Omron CX-Programmer project NewProject (CX-Programmer 9.73)

# PLC NewPLC1: C200HS CPU01

## Program NewProgram1 (no task)
; 欧姆龙电镀控制系统。 系统通过启动按钮启动工作流程，控制加热器、搅拌器和电镀电源，并包含故障检测和保护功能。 / 项目使用的物理设备包括PLC控制器、启动按钮、停止按钮、手动/自动开关、加热器、搅拌器、电镀电源、温度传感器、液位传感器、电流传感器和报警灯。 / 系统配备启动按钮、停止按钮和手动/自动切换开关。 / 在自动模式下，启动按钮触发系统运行。只有在停止按钮未按下时，系统才能启动，同时模式信号表示系统处于自动运行状态。 / 系统启动后，加热器开始工作。 / 搅拌器启动后，利用搅拌延时定时器 (TIM492) 控制搅拌时间。 / 电镀电源启动后，由电镀延时定时器 (TIM499) 控制电镀时长。 / 系统运行期间，监控关键参数。电流传感器将检测值与安全上限进行比较。液位传感器将检测值与安全下限进行比较。 / 当温度传感器检测到温度超出安全范围时，报警灯亮起。当电流传感器检测到电流超过安全上限时，报警灯亮起。当液位传感器检测到液位低于安全下限时，报警灯亮起。报警信号用于记录系统异常状态。 / 在手动模式下，操作员可控制设备。 / 实际应用中，该系统部署在电镀车间，使用的物理设备包括PLC控制器C200HS CPU01、启动按钮、停止按钮、手动/自动切换开关、加热器、搅拌器、电镀电源，以及温度传感器、液位传感器、电流传感器和报警灯。 / 为确保系统稳定运行，维护人员需定期检查温度传感器、液位传感器和电流传感器的工作状态，确认手动/自动切换开关切换正常，验证搅拌延时定时器 (TIM492) 和电镀延时定时器 (TIM499) 的时间设置是否准确，并通过观察报警灯的状态及时响应异常情况。 / 程序以END指令结束扫描周期，确保每次运行逻辑清晰可控。

### Section Section1

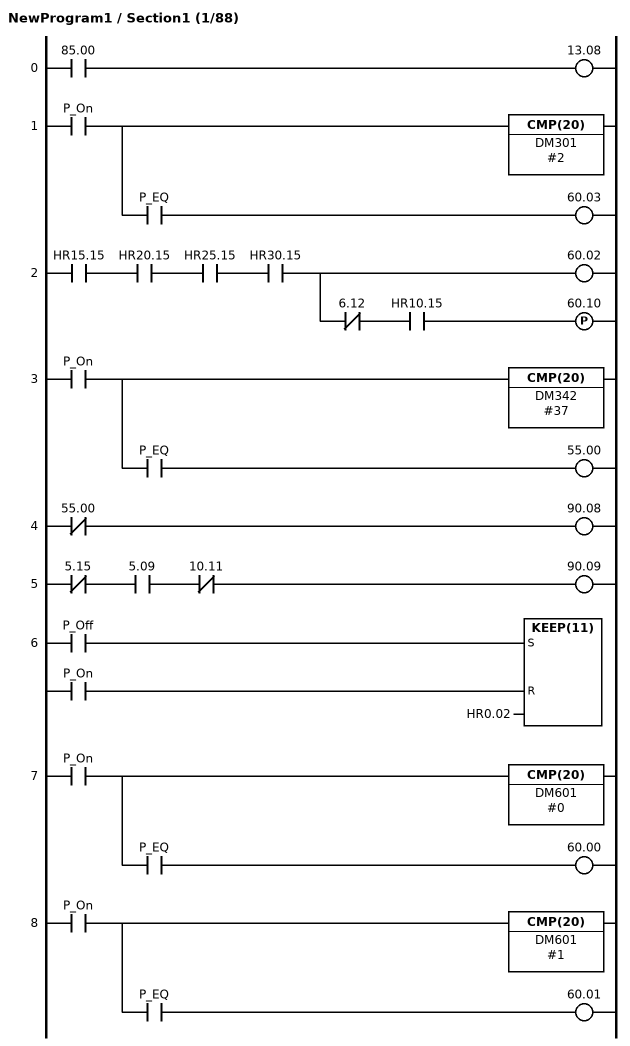
; rung 0
LD 85.00
OUT 13.08
; rung 1
LD P_On
CMP(20) DM301 #2
AND P_EQ
OUT 60.03
; rung 2
LD HR15.15
AND HR20.15
AND HR25.15
AND HR30.15
OUT 60.02
ANDNOT 6.12
AND HR10.15
DIFU(13) 60.10
; rung 3
LD P_On
CMP(20) DM342 #37
AND P_EQ
OUT 55.00
; rung 4
LDNOT 55.00
OUT 90.08
; rung 5
LDNOT 5.15
AND 5.09
ANDNOT 10.11
OUT 90.09
; rung 6
LD P_Off
LD P_On
KEEP(11) HR0.02
; rung 7
LD P_On
CMP(20) DM601 #0
AND P_EQ
OUT 60.00
; rung 8
LD P_On
CMP(20) DM601 #1
AND P_EQ
OUT 60.01

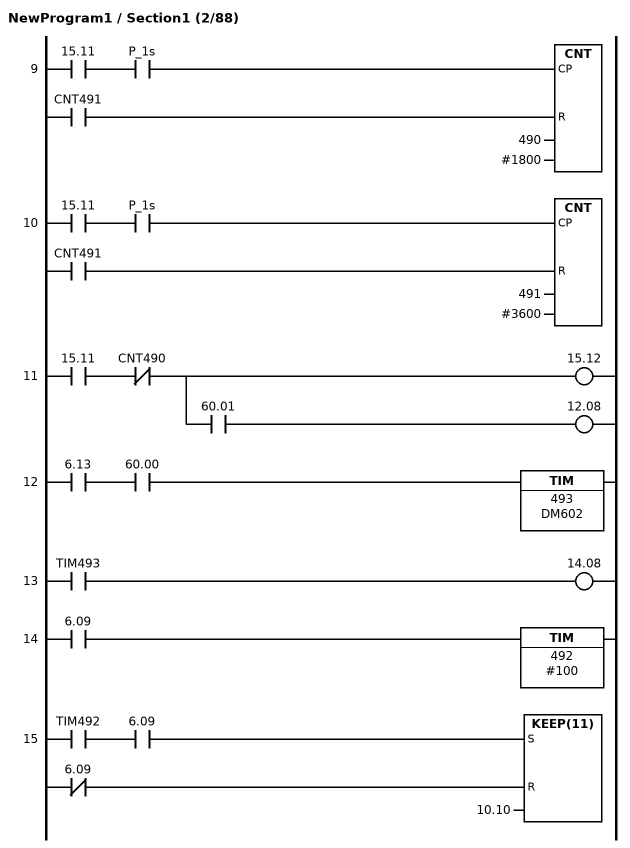
; rung 9
LD 15.11
AND P_1s
LD CNT491
CNT 490 #1800
; rung 10
LD 15.11
AND P_1s
LD CNT491
CNT 491 #3600
; rung 11
LD 15.11
ANDNOT CNT490
OUT 15.12
AND 60.01
OUT 12.08
; rung 12
LD 6.13
AND 60.00
TIM 493 DM602
; rung 13
LD TIM493
OUT 14.08
; rung 14
LD 6.09
TIM 492 #100
; rung 15
LD TIM492
AND 6.09
LDNOT 6.09
KEEP(11) 10.10

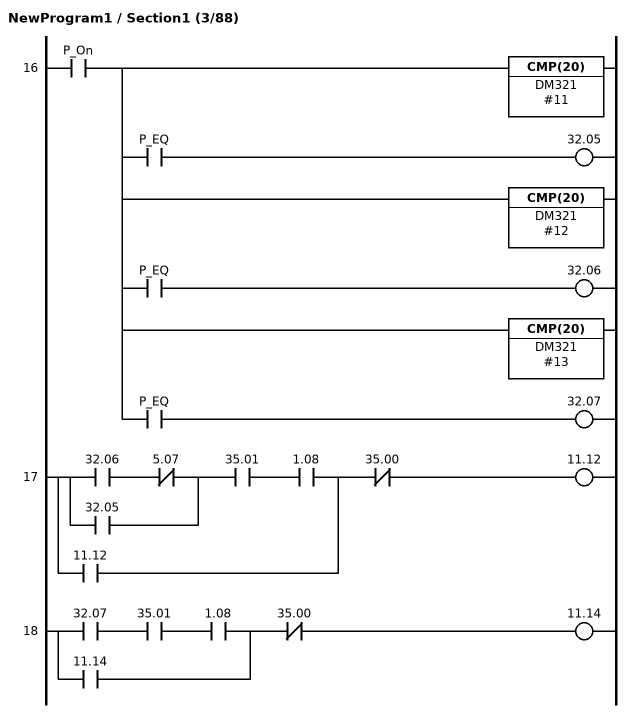
; rung 16
LD P_On
OUT TR0
CMP(20) DM321 #11
AND P_EQ
OUT 32.05
LD TR0
CMP(20) DM321 #12
AND P_EQ
OUT 32.06
LD TR0
CMP(20) DM321 #13
AND P_EQ
OUT 32.07
; rung 17
LD 32.06
ANDNOT 5.07
OR 32.05
AND 35.01
AND 1.08
OR 11.12
ANDNOT 35.00
OUT 11.12
; rung 18
LD 32.07
AND 35.01
AND 1.08
OR 11.14
ANDNOT 35.00
OUT 11.14

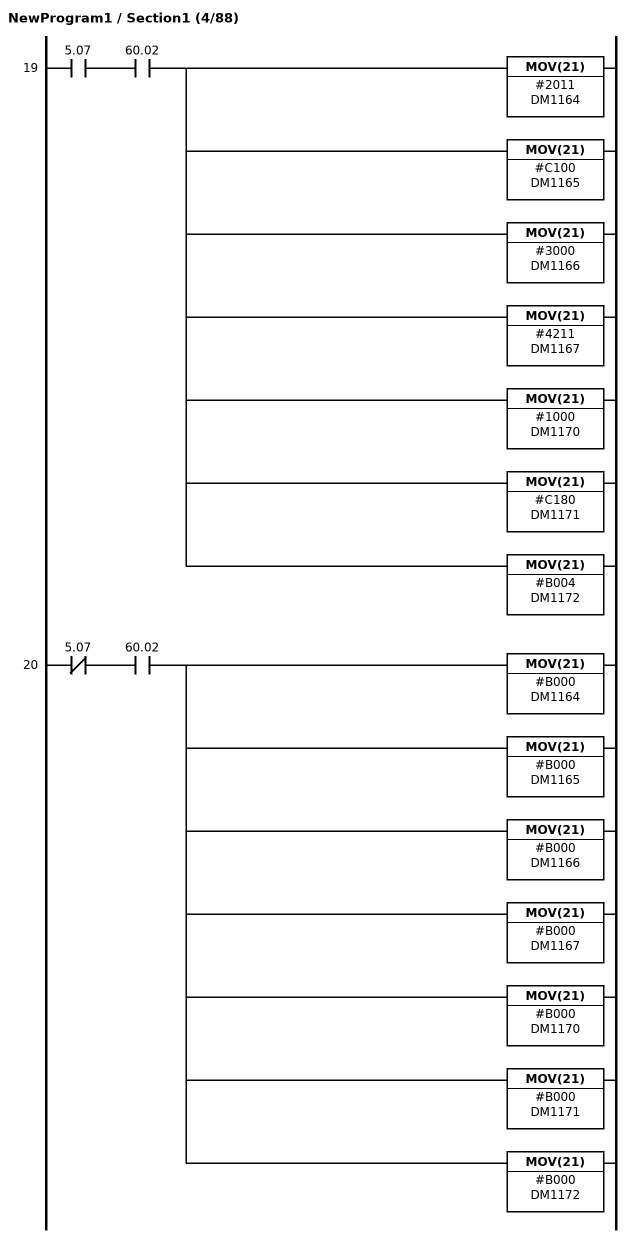
; rung 19
LD 5.07
AND 60.02
MOV(21) #2011 DM1164
MOV(21) #C100 DM1165
MOV(21) #3000 DM1166
MOV(21) #4211 DM1167
MOV(21) #1000 DM1170
MOV(21) #C180 DM1171
MOV(21) #B004 DM1172
; rung 20
LDNOT 5.07
AND 60.02
MOV(21) #B000 DM1164
MOV(21) #B000 DM1165
MOV(21) #B000 DM1166
MOV(21) #B000 DM1167
MOV(21) #B000 DM1170
MOV(21) #B000 DM1171
MOV(21) #B000 DM1172

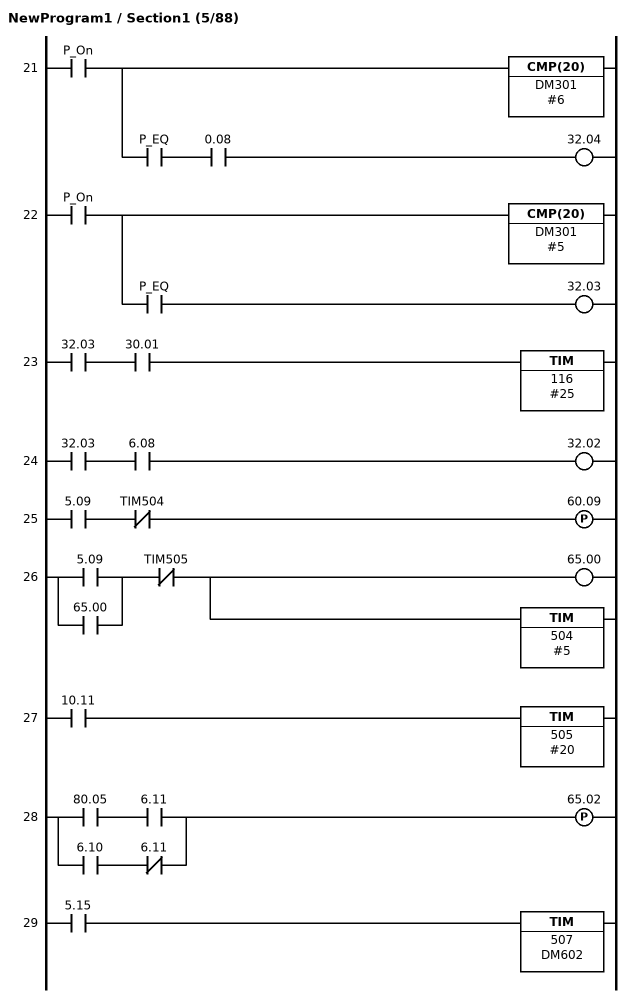
; rung 21
LD P_On
CMP(20) DM301 #6
AND P_EQ
AND 0.08
OUT 32.04
; rung 22
LD P_On
CMP(20) DM301 #5
AND P_EQ
OUT 32.03
; rung 23
LD 32.03
AND 30.01
TIM 116 #25
; rung 24
LD 32.03
AND 6.08
OUT 32.02
; rung 25
LD 5.09
ANDNOT TIM504
DIFU(13) 60.09
; rung 26
LD 5.09
OR 65.00
ANDNOT TIM505
OUT 65.00
TIM 504 #5
; rung 27
LD 10.11
TIM 505 #20
; rung 28
LD 80.05
AND 6.11
LD 6.10
ANDNOT 6.11
ORLD
DIFU(13) 65.02
; rung 29
LD 5.15
TIM 507 DM602

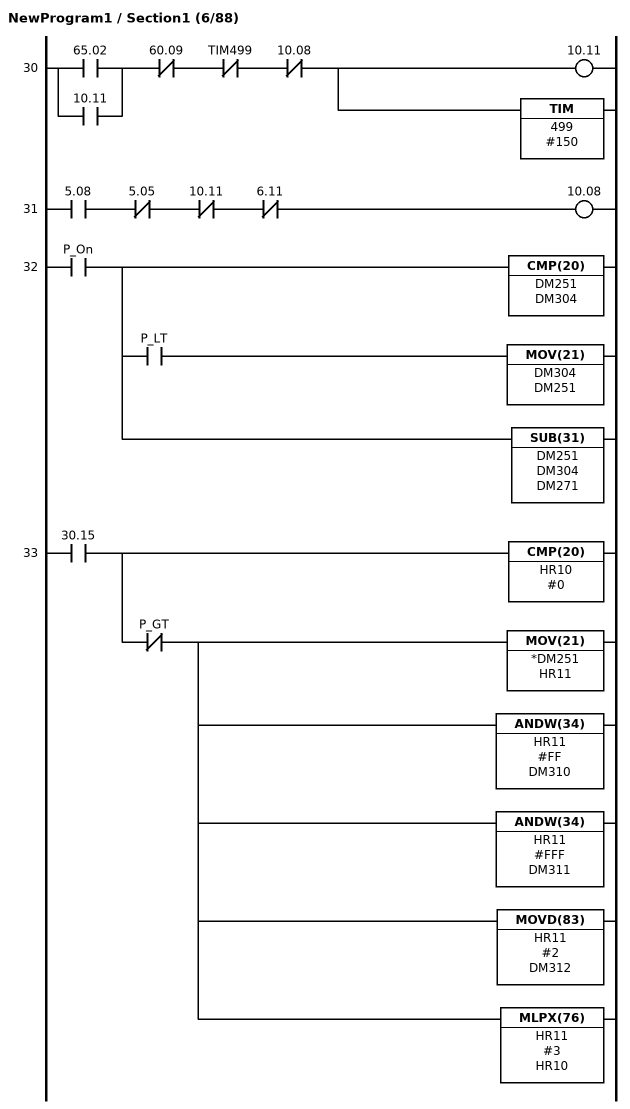
; rung 30
LD 65.02
OR 10.11
ANDNOT 60.09
ANDNOT TIM499
ANDNOT 10.08
OUT 10.11
TIM 499 #150
; rung 31
LD 5.08
ANDNOT 5.05
ANDNOT 10.11
ANDNOT 6.11
OUT 10.08
; rung 32
LD P_On
OUT TR0
CMP(20) DM251 DM304
AND P_LT
MOV(21) DM304 DM251
LD TR0
SUB(31) DM251 DM304 DM271
; rung 33
LD 30.15
CMP(20) HR10 #0
ANDNOT P_GT
MOV(21) *DM251 HR11
ANDW(34) HR11 #FF DM310
ANDW(34) HR11 #FFF DM311
MOVD(83) HR11 #2 DM312
MLPX(76) HR11 #3 HR10

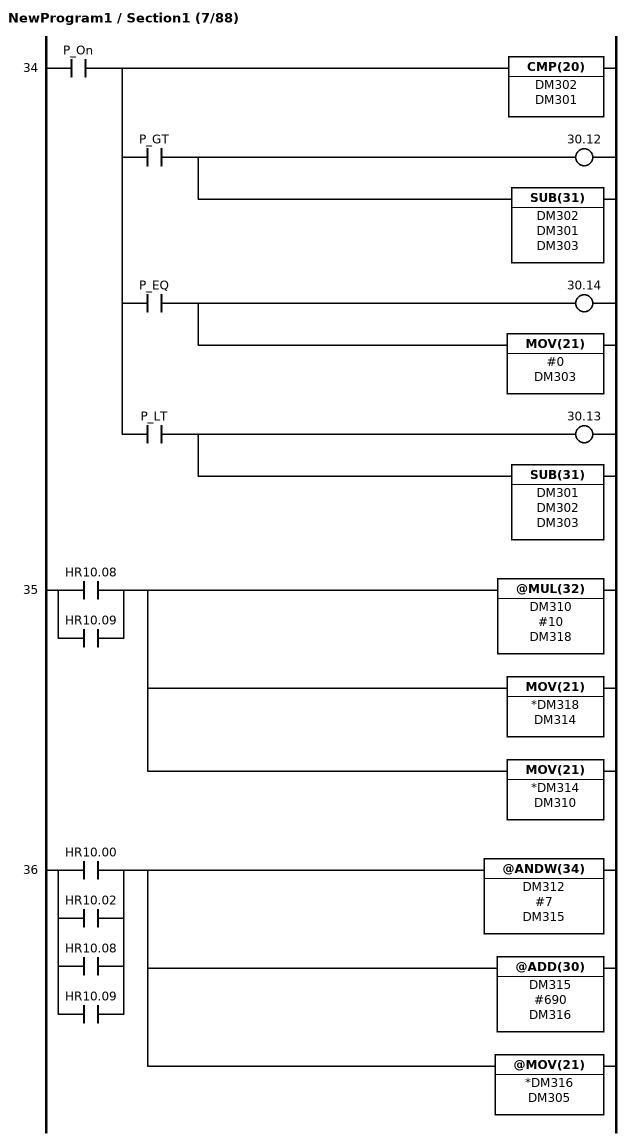
; rung 34
LD P_On
OUT TR0
CMP(20) DM302 DM301
AND P_GT
OUT 30.12
SUB(31) DM302 DM301 DM303
LD TR0
AND P_EQ
OUT 30.14
MOV(21) #0 DM303
LD TR0
AND P_LT
OUT 30.13
SUB(31) DM301 DM302 DM303
; rung 35
LD HR10.08
OR HR10.09
@MUL(32) DM310 #10 DM318
MOV(21) *DM318 DM314
MOV(21) *DM314 DM310
; rung 36
LD HR10.00
OR HR10.02
OR HR10.08
OR HR10.09
@ANDW(34) DM312 #7 DM315
@ADD(30) DM315 #690 DM316
@MOV(21) *DM316 DM305

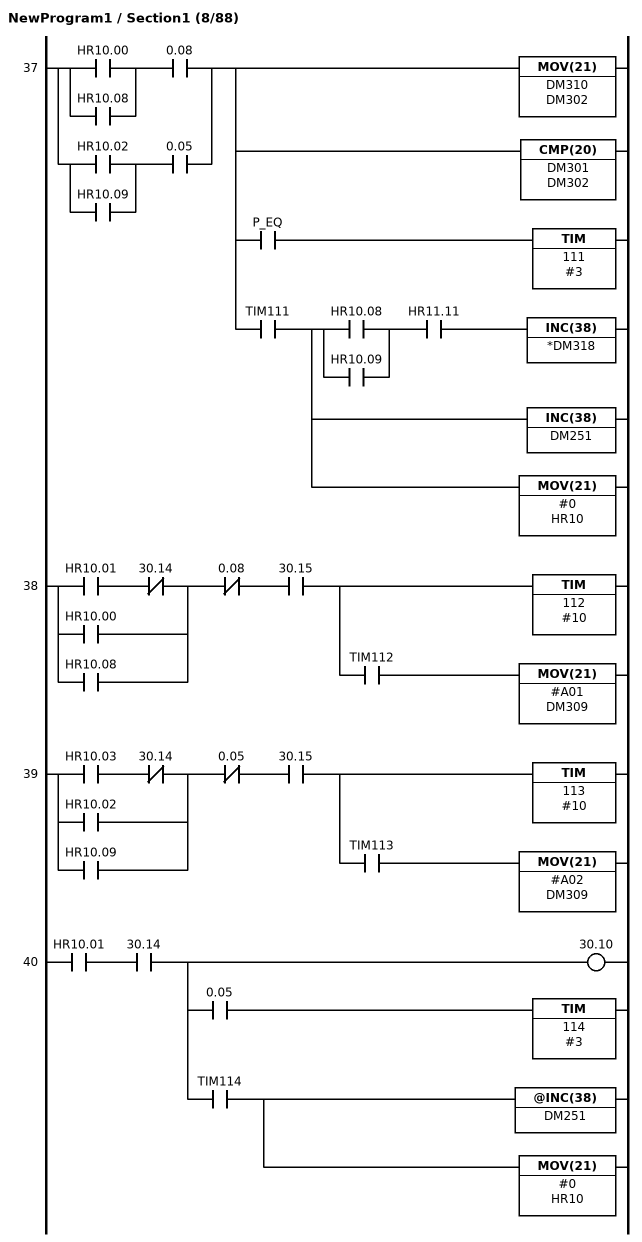
; rung 37
LD HR10.00
OR HR10.08
AND 0.08
LD HR10.02
OR HR10.09
AND 0.05
ORLD
OUT TR0
MOV(21) DM310 DM302
CMP(20) DM301 DM302
AND P_EQ
TIM 111 #3
LD TR0
AND TIM111
OUT TR0
LD HR10.08
OR HR10.09
ANDLD
AND HR11.11
INC(38) *DM318
LD TR0
INC(38) DM251
MOV(21) #0 HR10
; rung 38
LD HR10.01
ANDNOT 30.14
OR HR10.00
OR HR10.08
ANDNOT 0.08
AND 30.15
TIM 112 #10
AND TIM112
MOV(21) #A01 DM309
; rung 39
LD HR10.03
ANDNOT 30.14
OR HR10.02
OR HR10.09
ANDNOT 0.05
AND 30.15
TIM 113 #10
AND TIM113
MOV(21) #A02 DM309
; rung 40
LD HR10.01
AND 30.14
OUT TR0
OUT 30.10
AND 0.05
TIM 114 #3
LD TR0
AND TIM114
@INC(38) DM251
MOV(21) #0 HR10

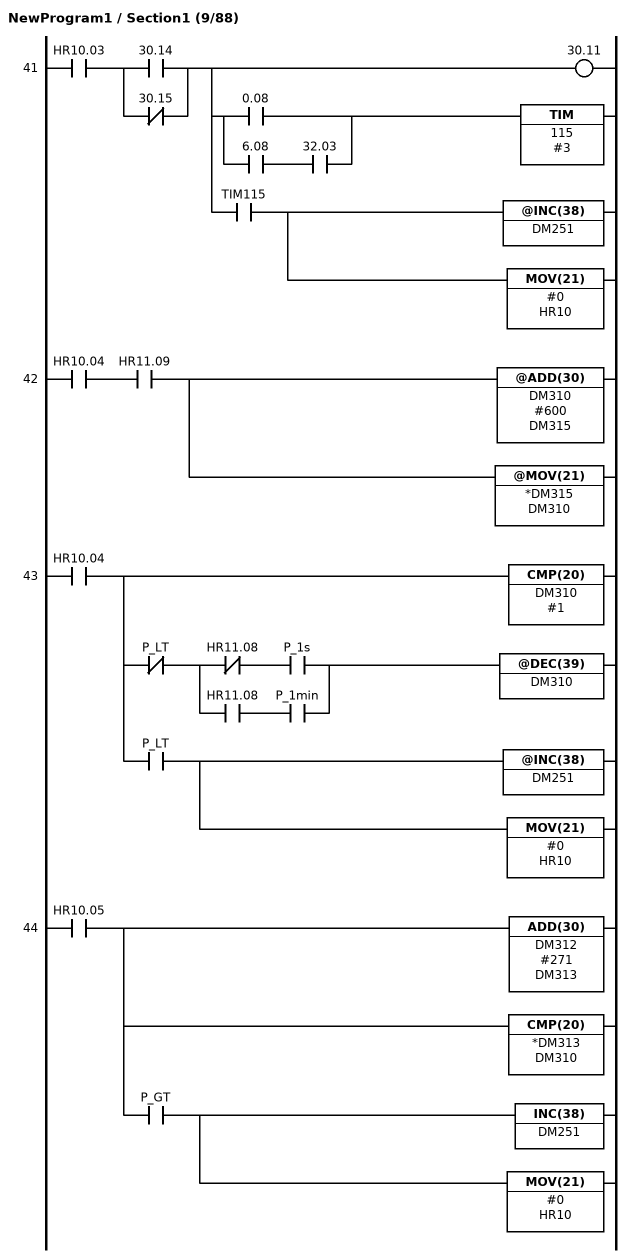
; rung 41
LD HR10.03
LD 30.14
ORNOT 30.15
ANDLD
OUT TR0
OUT 30.11
LD 0.08
LD 6.08
AND 32.03
ORLD
ANDLD
TIM 115 #3
LD TR0
AND TIM115
@INC(38) DM251
MOV(21) #0 HR10
; rung 42
LD HR10.04
AND HR11.09
@ADD(30) DM310 #600 DM315
@MOV(21) *DM315 DM310
; rung 43
LD HR10.04
OUT TR0
CMP(20) DM310 #1
ANDNOT P_LT
LDNOT HR11.08
AND P_1s
LD HR11.08
AND P_1min
ORLD
ANDLD
@DEC(39) DM310
LD TR0
AND P_LT
@INC(38) DM251
MOV(21) #0 HR10
; rung 44
LD HR10.05
ADD(30) DM312 #271 DM313
CMP(20) *DM313 DM310
AND P_GT
INC(38) DM251
MOV(21) #0 HR10

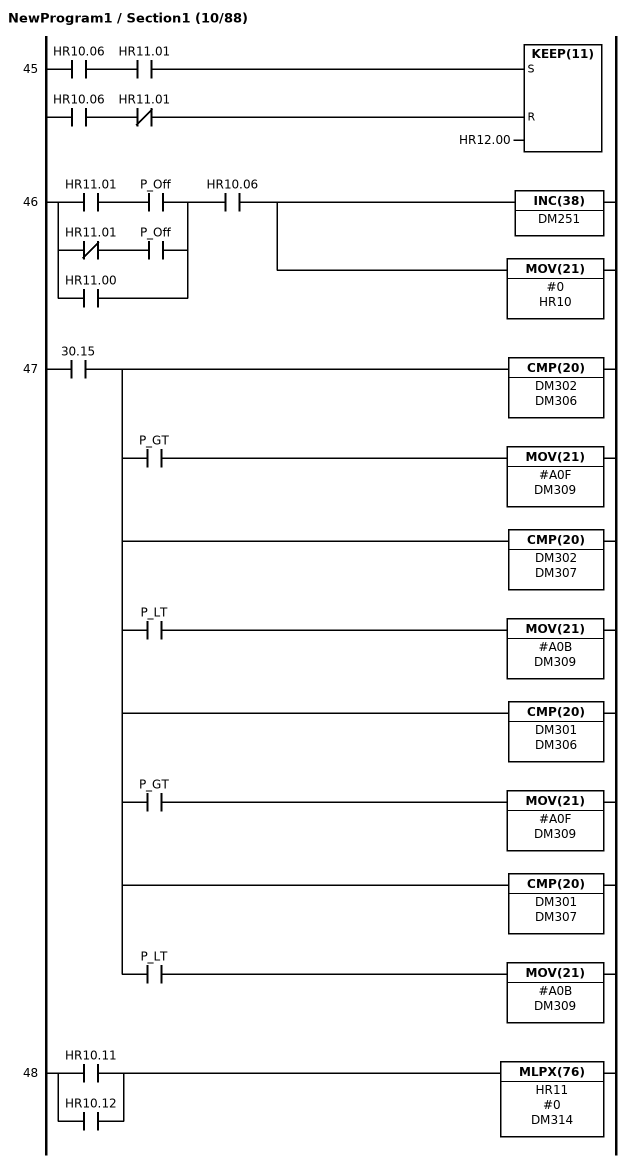
; rung 45
LD HR10.06
AND HR11.01
LD HR10.06
ANDNOT HR11.01
KEEP(11) HR12.00
; rung 46
LD HR11.01
AND P_Off
LDNOT HR11.01
AND P_Off
ORLD
OR HR11.00
AND HR10.06
INC(38) DM251
MOV(21) #0 HR10
; rung 47
LD 30.15
OUT TR0
CMP(20) DM302 DM306
AND P_GT
MOV(21) #A0F DM309
LD TR0
CMP(20) DM302 DM307
AND P_LT
MOV(21) #A0B DM309
LD TR0
CMP(20) DM301 DM306
AND P_GT
MOV(21) #A0F DM309
LD TR0
CMP(20) DM301 DM307
AND P_LT
MOV(21) #A0B DM309
; rung 48
LD HR10.11
OR HR10.12
MLPX(76) HR11 #0 DM314

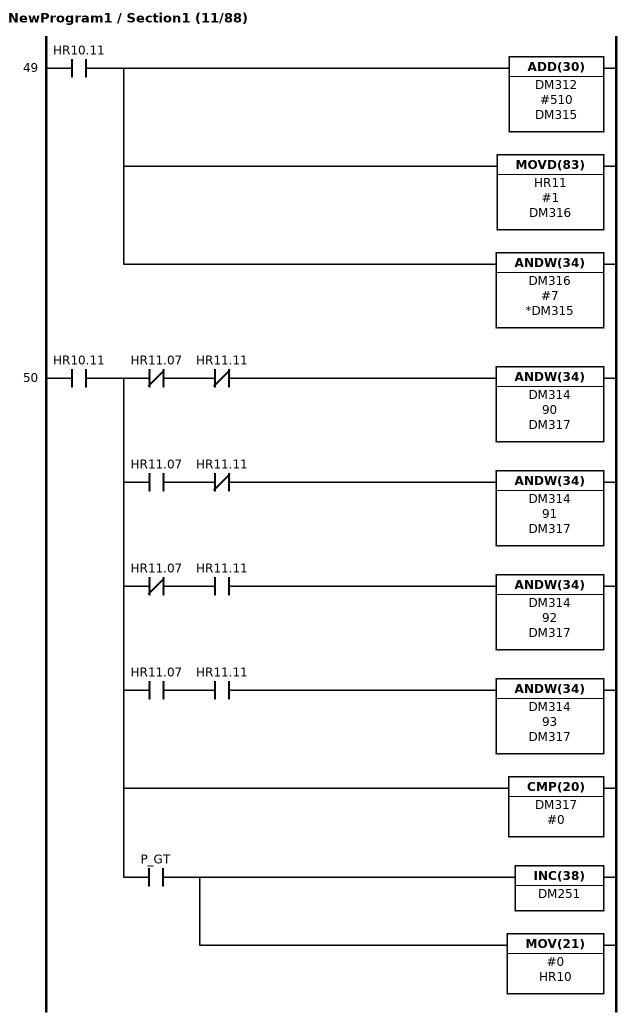
; rung 49
LD HR10.11
ADD(30) DM312 #510 DM315
MOVD(83) HR11 #1 DM316
ANDW(34) DM316 #7 *DM315
; rung 50
LD HR10.11
OUT TR0
ANDNOT HR11.07
ANDNOT HR11.11
ANDW(34) DM314 90 DM317
LD TR0
AND HR11.07
ANDNOT HR11.11
ANDW(34) DM314 91 DM317
LD TR0
ANDNOT HR11.07
AND HR11.11
ANDW(34) DM314 92 DM317
LD TR0
AND HR11.07
AND HR11.11
ANDW(34) DM314 93 DM317
LD TR0
CMP(20) DM317 #0
AND P_GT
INC(38) DM251
MOV(21) #0 HR10

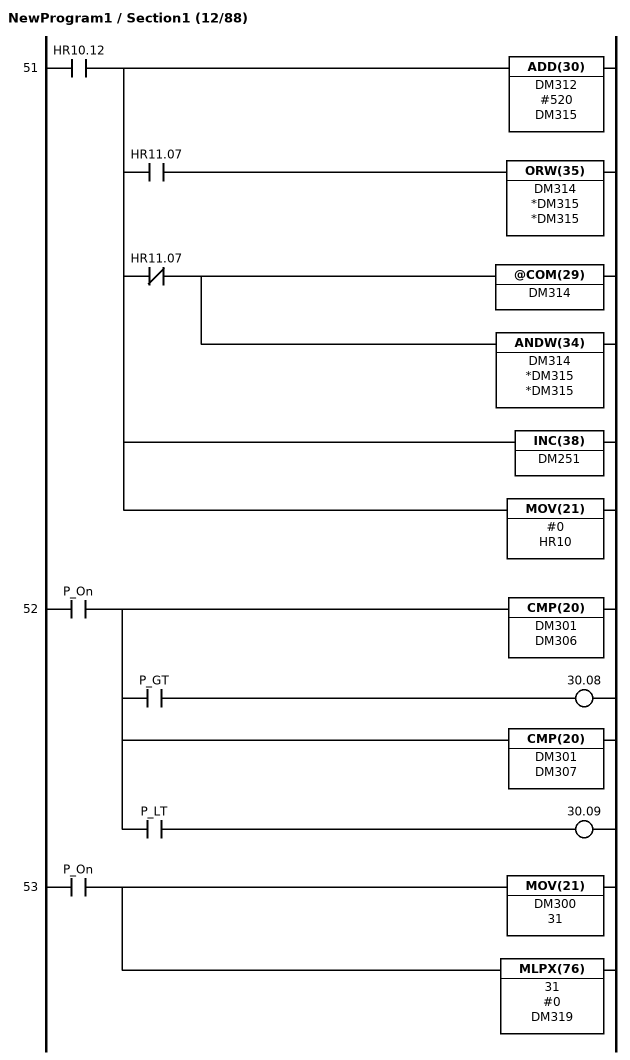
; rung 51
LD HR10.12
OUT TR0
ADD(30) DM312 #520 DM315
AND HR11.07
ORW(35) DM314 *DM315 *DM315
LD TR0
ANDNOT HR11.07
@COM(29) DM314
ANDW(34) DM314 *DM315 *DM315
LD TR0
INC(38) DM251
MOV(21) #0 HR10
; rung 52
LD P_On
OUT TR0
CMP(20) DM301 DM306
AND P_GT
OUT 30.08
LD TR0
CMP(20) DM301 DM307
AND P_LT
OUT 30.09
; rung 53
LD P_On
MOV(21) DM300 31
MLPX(76) 31 #0 DM319

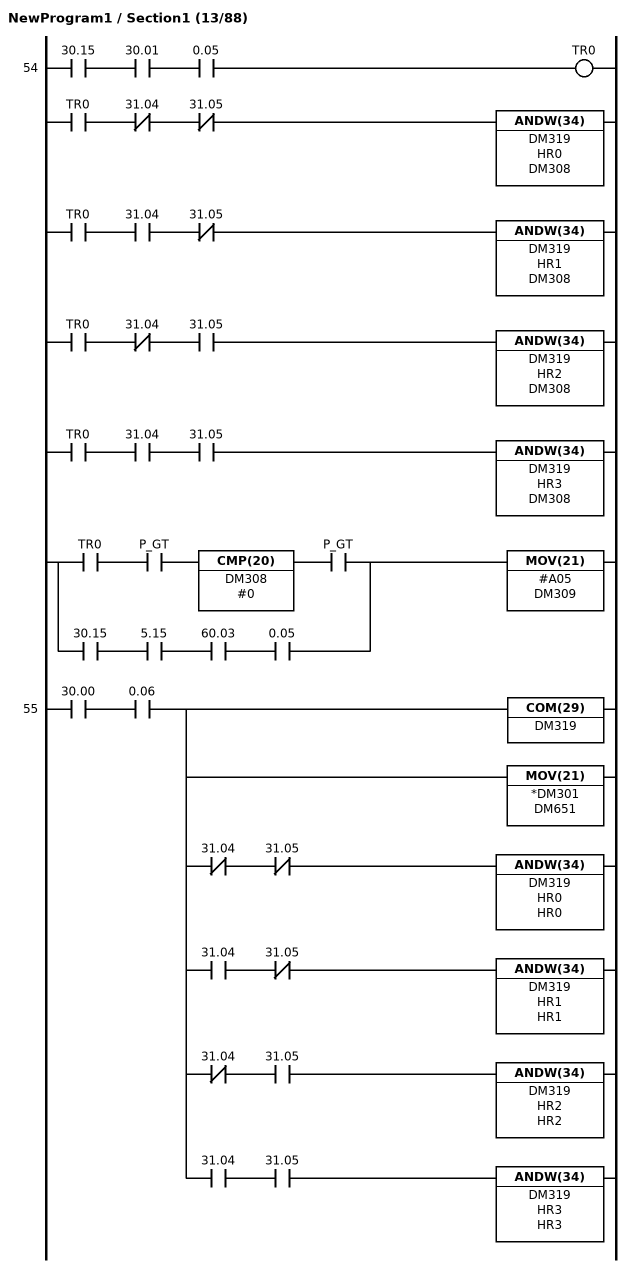
; rung 54
LD 30.15
AND 30.01
AND 0.05
OUT TR0
ANDNOT 31.04
ANDNOT 31.05
ANDW(34) DM319 HR0 DM308
LD TR0
AND 31.04
ANDNOT 31.05
ANDW(34) DM319 HR1 DM308
LD TR0
ANDNOT 31.04
AND 31.05
ANDW(34) DM319 HR2 DM308
LD TR0
AND 31.04
AND 31.05
ANDW(34) DM319 HR3 DM308
LD TR0
AND P_GT
CMP(20) DM308 #0
AND P_GT
LD 30.15
AND 5.15
AND 60.03
AND 0.05
ORLD
MOV(21) #A05 DM309
; rung 55
LD 30.00
AND 0.06
OUT TR0
COM(29) DM319
MOV(21) *DM301 DM651
ANDNOT 31.04
ANDNOT 31.05
ANDW(34) DM319 HR0 HR0
LD TR0
AND 31.04
ANDNOT 31.05
ANDW(34) DM319 HR1 HR1
LD TR0
ANDNOT 31.04
AND 31.05
ANDW(34) DM319 HR2 HR2
LD TR0
AND 31.04
AND 31.05
ANDW(34) DM319 HR3 HR3

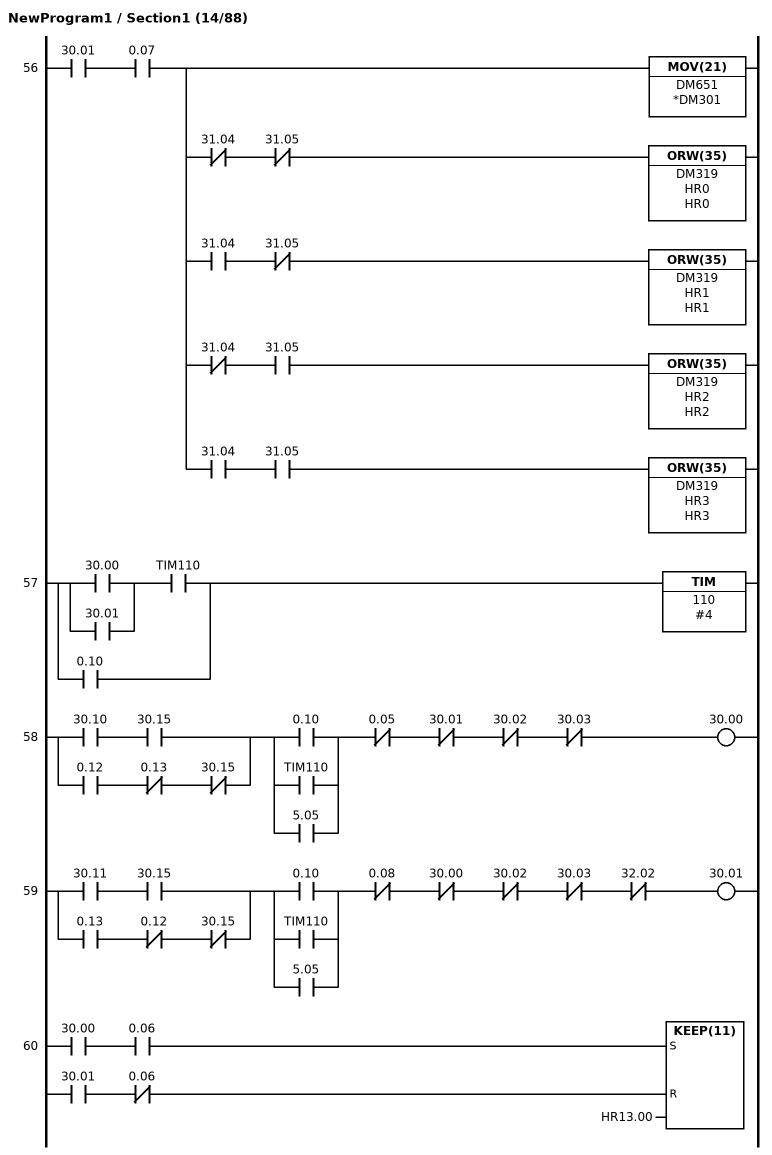
; rung 56
LD 30.01
AND 0.07
OUT TR0
MOV(21) DM651 *DM301
ANDNOT 31.04
ANDNOT 31.05
ORW(35) DM319 HR0 HR0
LD TR0
AND 31.04
ANDNOT 31.05
ORW(35) DM319 HR1 HR1
LD TR0
ANDNOT 31.04
AND 31.05
ORW(35) DM319 HR2 HR2
LD TR0
AND 31.04
AND 31.05
ORW(35) DM319 HR3 HR3
; rung 57
LD 30.00
OR 30.01
AND TIM110
OR 0.10
TIM 110 #4
; rung 58
LD 30.10
AND 30.15
LD 0.12
ANDNOT 0.13
ANDNOT 30.15
ORLD
LD 0.10
OR TIM110
OR 5.05
ANDLD
ANDNOT 0.05
ANDNOT 30.01
ANDNOT 30.02
ANDNOT 30.03
OUT 30.00
; rung 59
LD 30.11
AND 30.15
LD 0.13
ANDNOT 0.12
ANDNOT 30.15
ORLD
LD 0.10
OR TIM110
OR 5.05
ANDLD
ANDNOT 0.08
ANDNOT 30.00
ANDNOT 30.02
ANDNOT 30.03
ANDNOT 32.02
OUT 30.01
; rung 60
LD 30.00
AND 0.06
LD 30.01
ANDNOT 0.06
KEEP(11) HR13.00

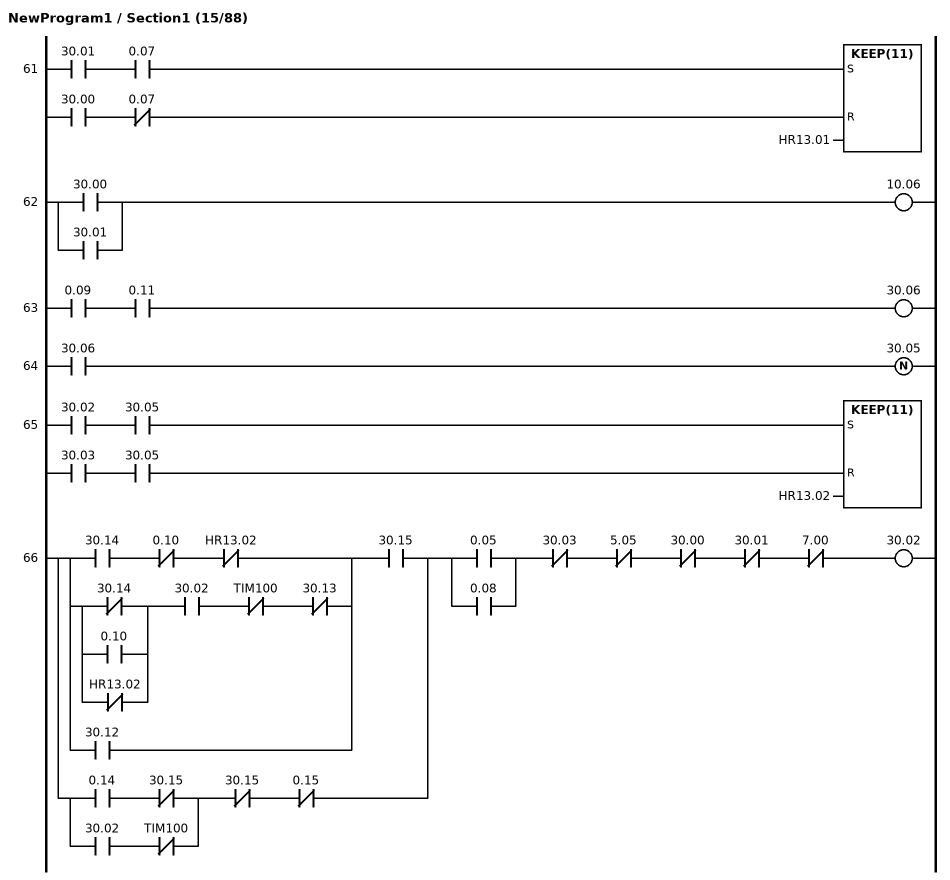
; rung 61
LD 30.01
AND 0.07
LD 30.00
ANDNOT 0.07
KEEP(11) HR13.01
; rung 62
LD 30.00
OR 30.01
OUT 10.06
; rung 63
LD 0.09
AND 0.11
OUT 30.06
; rung 64
LD 30.06
DIFD(14) 30.05
; rung 65
LD 30.02
AND 30.05
LD 30.03
AND 30.05
KEEP(11) HR13.02
; rung 66
LD 30.14
ANDNOT 0.10
ANDNOT HR13.02
LDNOT 30.14
OR 0.10
ORNOT HR13.02
AND 30.02
ANDNOT TIM100
ANDNOT 30.13
ORLD
OR 30.12
AND 30.15
LD 0.14
ANDNOT 30.15
LD 30.02
ANDNOT TIM100
ORLD
ANDNOT 30.15
ANDNOT 0.15
ORLD
LD 0.05
OR 0.08
ANDLD
ANDNOT 30.03
ANDNOT 5.05
ANDNOT 30.00
ANDNOT 30.01
ANDNOT 7.00
OUT 30.02

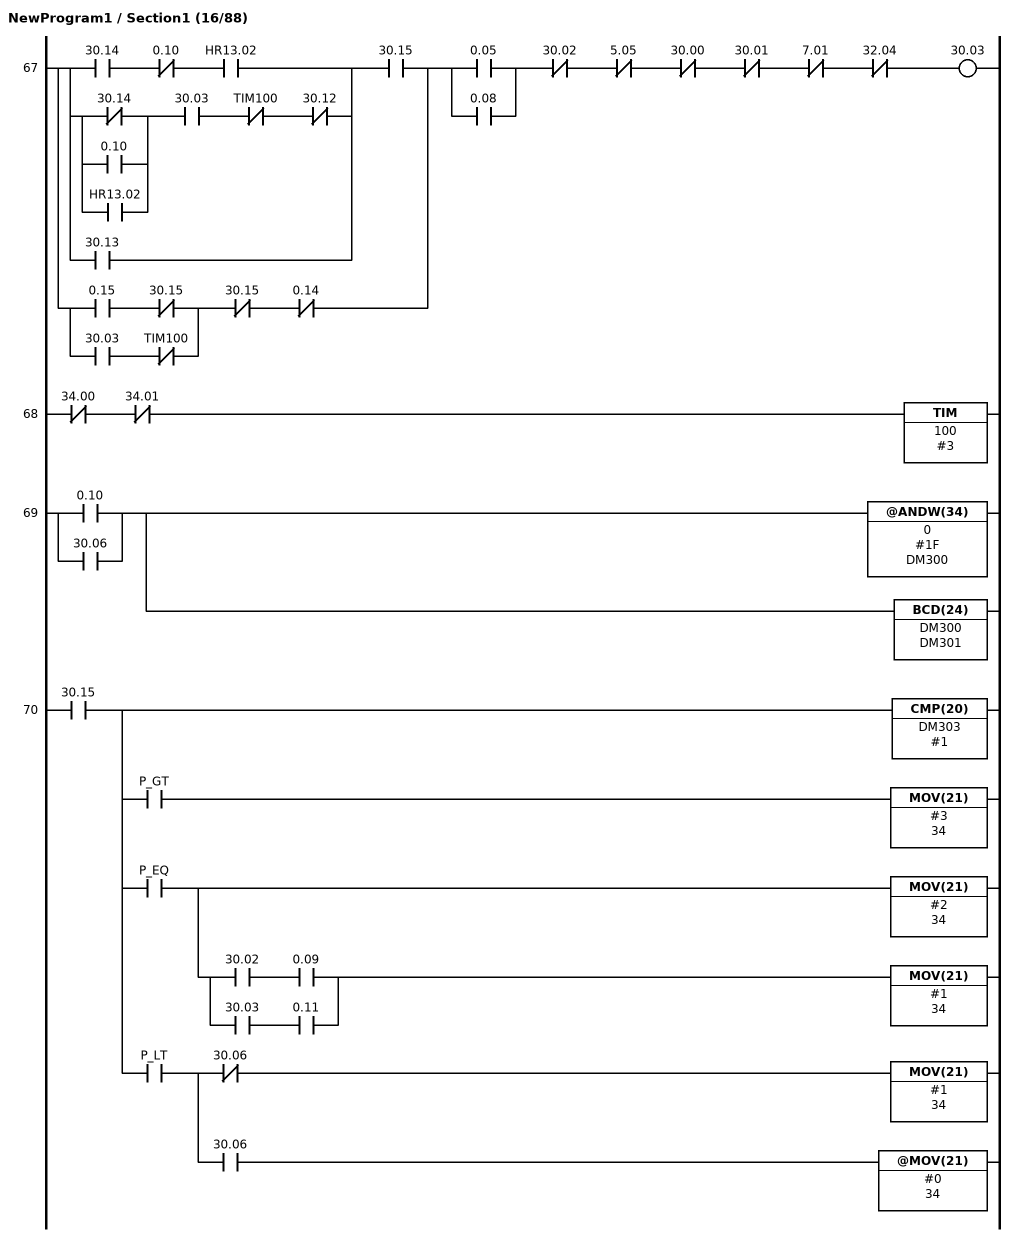
; rung 67
LD 30.14
ANDNOT 0.10
AND HR13.02
LDNOT 30.14
OR 0.10
OR HR13.02
AND 30.03
ANDNOT TIM100
ANDNOT 30.12
ORLD
OR 30.13
AND 30.15
LD 0.15
ANDNOT 30.15
LD 30.03
ANDNOT TIM100
ORLD
ANDNOT 30.15
ANDNOT 0.14
ORLD
LD 0.05
OR 0.08
ANDLD
ANDNOT 30.02
ANDNOT 5.05
ANDNOT 30.00
ANDNOT 30.01
ANDNOT 7.01
ANDNOT 32.04
OUT 30.03
; rung 68
LDNOT 34.00
ANDNOT 34.01
TIM 100 #3
; rung 69
LD 0.10
OR 30.06
@ANDW(34) 0 #1F DM300
BCD(24) DM300 DM301
; rung 70
LD 30.15
OUT TR0
CMP(20) DM303 #1
AND P_GT
MOV(21) #3 34
LD TR0
AND P_EQ
MOV(21) #2 34
LD 30.02
AND 0.09
LD 30.03
AND 0.11
ORLD
ANDLD
MOV(21) #1 34
LD TR0
AND P_LT
OUT TR0
ANDNOT 30.06
MOV(21) #1 34
LD TR0
AND 30.06
@MOV(21) #0 34

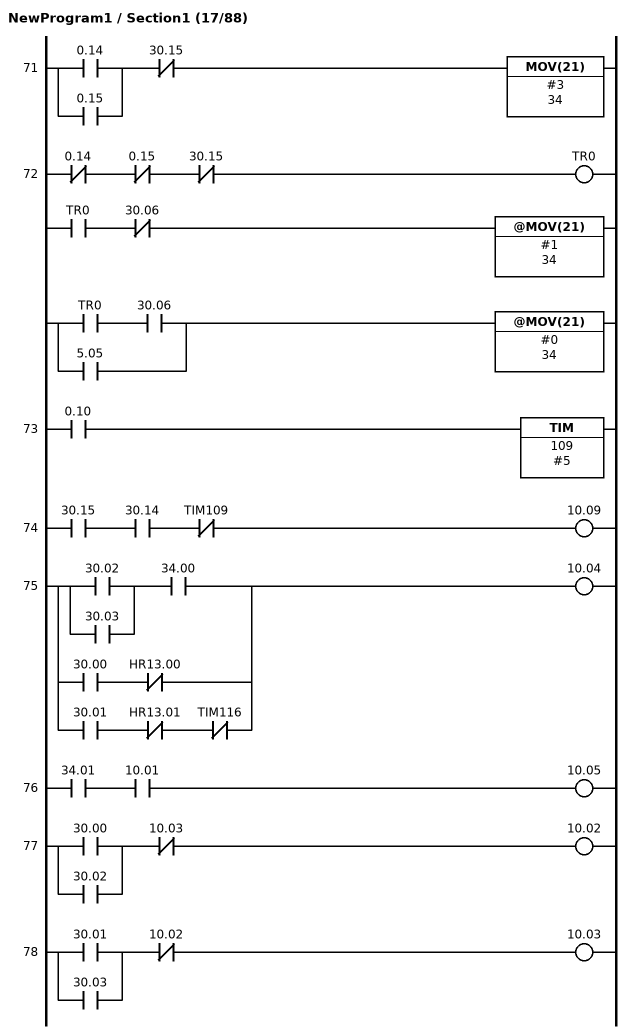
; rung 71
LD 0.14
OR 0.15
ANDNOT 30.15
MOV(21) #3 34
; rung 72
LDNOT 0.14
ANDNOT 0.15
ANDNOT 30.15
OUT TR0
ANDNOT 30.06
@MOV(21) #1 34
LD TR0
AND 30.06
OR 5.05
@MOV(21) #0 34
; rung 73
LD 0.10
TIM 109 #5
; rung 74
LD 30.15
AND 30.14
ANDNOT TIM109
OUT 10.09
; rung 75
LD 30.02
OR 30.03
AND 34.00
LD 30.00
ANDNOT HR13.00
ORLD
LD 30.01
ANDNOT HR13.01
ANDNOT TIM116
ORLD
OUT 10.04
; rung 76
LD 34.01
AND 10.01
OUT 10.05
; rung 77
LD 30.00
OR 30.02
ANDNOT 10.03
OUT 10.02
; rung 78
LD 30.01
OR 30.03
ANDNOT 10.02
OUT 10.03

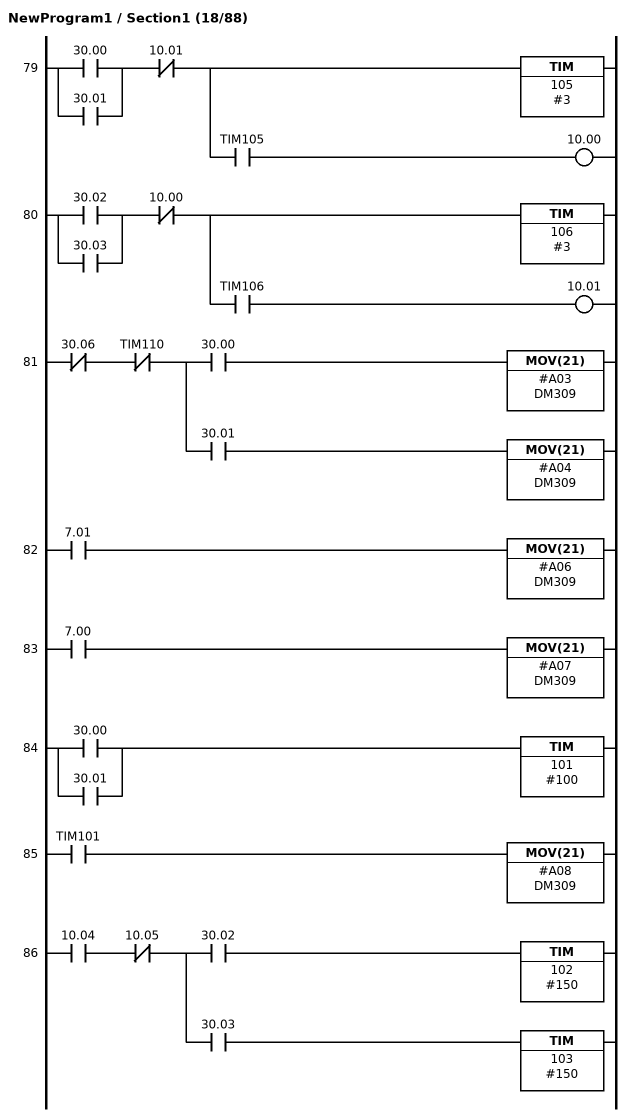
; rung 79
LD 30.00
OR 30.01
ANDNOT 10.01
TIM 105 #3
AND TIM105
OUT 10.00
; rung 80
LD 30.02
OR 30.03
ANDNOT 10.00
TIM 106 #3
AND TIM106
OUT 10.01
; rung 81
LDNOT 30.06
ANDNOT TIM110
OUT TR0
AND 30.00
MOV(21) #A03 DM309
LD TR0
AND 30.01
MOV(21) #A04 DM309
; rung 82
LD 7.01
MOV(21) #A06 DM309
; rung 83
LD 7.00
MOV(21) #A07 DM309
; rung 84
LD 30.00
OR 30.01
TIM 101 #100
; rung 85
LD TIM101
MOV(21) #A08 DM309
; rung 86
LD 10.04
ANDNOT 10.05
OUT TR0
AND 30.02
TIM 102 #150
LD TR0
AND 30.03
TIM 103 #150

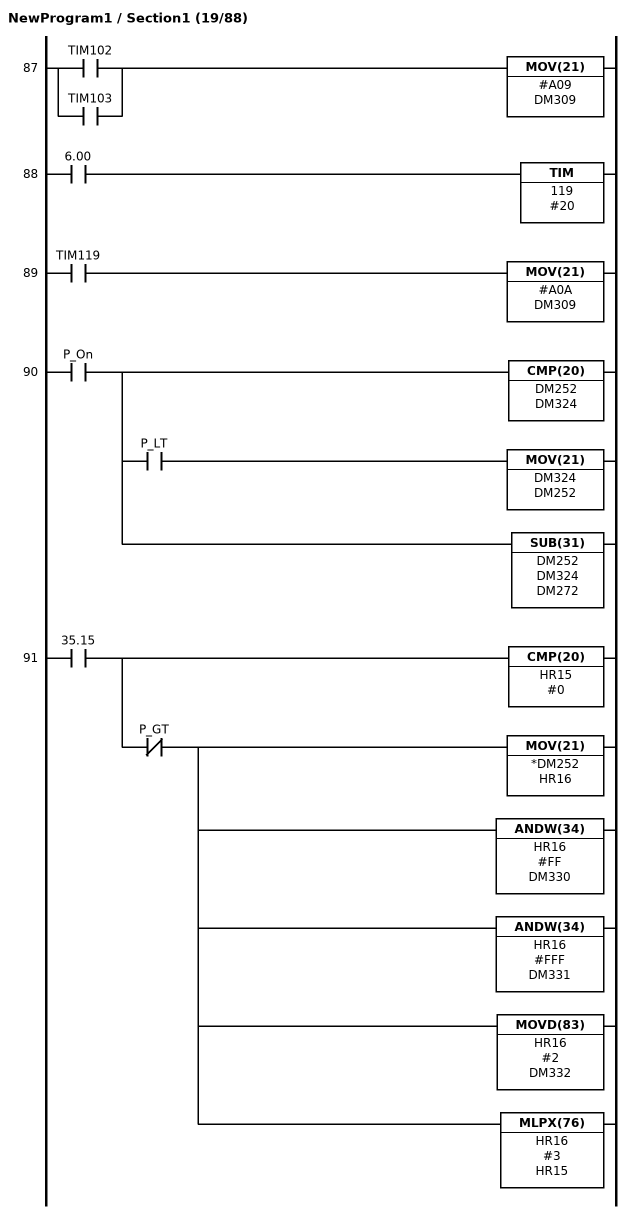
; rung 87
LD TIM102
OR TIM103
MOV(21) #A09 DM309
; rung 88
LD 6.00
TIM 119 #20
; rung 89
LD TIM119
MOV(21) #A0A DM309
; rung 90
LD P_On
OUT TR0
CMP(20) DM252 DM324
AND P_LT
MOV(21) DM324 DM252
LD TR0
SUB(31) DM252 DM324 DM272
; rung 91
LD 35.15
CMP(20) HR15 #0
ANDNOT P_GT
MOV(21) *DM252 HR16
ANDW(34) HR16 #FF DM330
ANDW(34) HR16 #FFF DM331
MOVD(83) HR16 #2 DM332
MLPX(76) HR16 #3 HR15

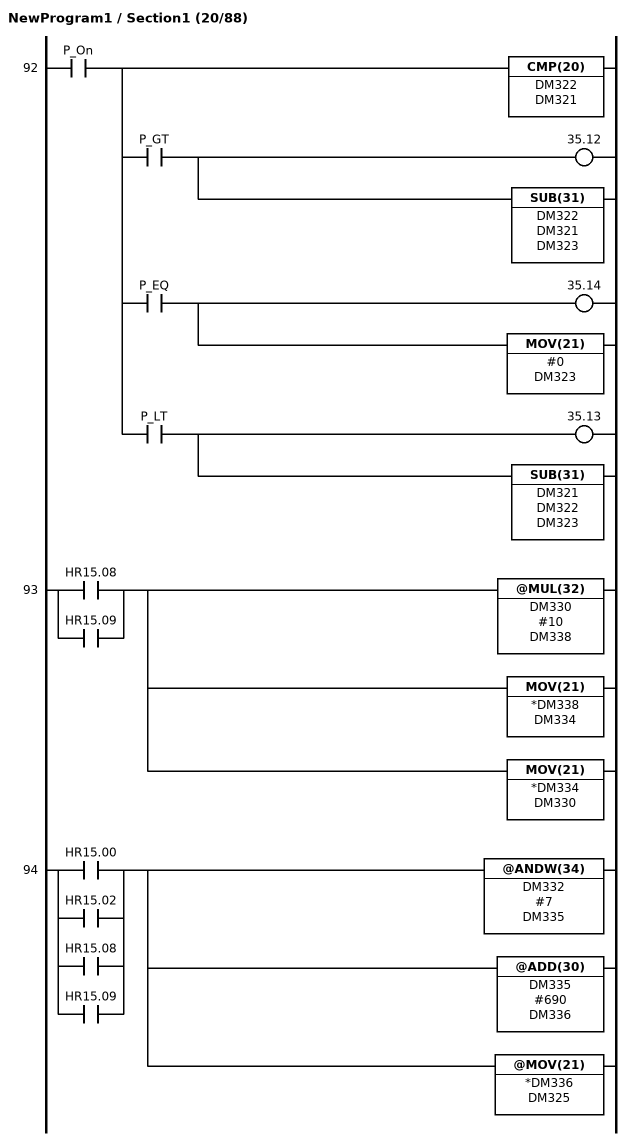
; rung 92
LD P_On
OUT TR0
CMP(20) DM322 DM321
AND P_GT
OUT 35.12
SUB(31) DM322 DM321 DM323
LD TR0
AND P_EQ
OUT 35.14
MOV(21) #0 DM323
LD TR0
AND P_LT
OUT 35.13
SUB(31) DM321 DM322 DM323
; rung 93
LD HR15.08
OR HR15.09
@MUL(32) DM330 #10 DM338
MOV(21) *DM338 DM334
MOV(21) *DM334 DM330
; rung 94
LD HR15.00
OR HR15.02
OR HR15.08
OR HR15.09
@ANDW(34) DM332 #7 DM335
@ADD(30) DM335 #690 DM336
@MOV(21) *DM336 DM325

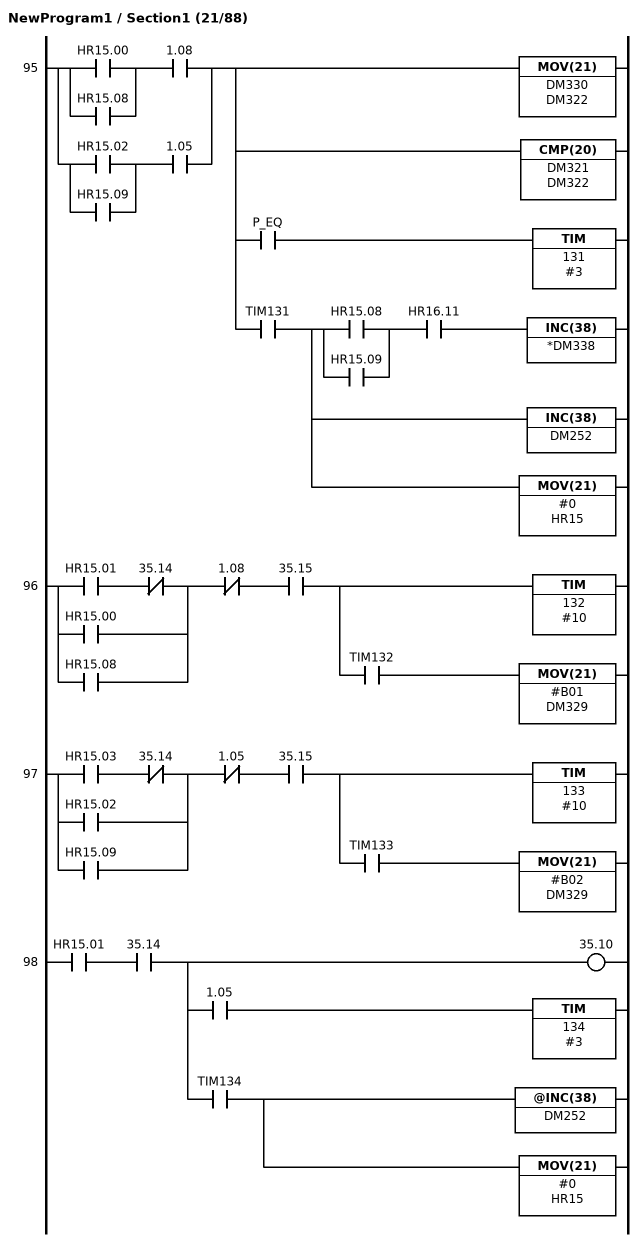
; rung 95
LD HR15.00
OR HR15.08
AND 1.08
LD HR15.02
OR HR15.09
AND 1.05
ORLD
OUT TR0
MOV(21) DM330 DM322
CMP(20) DM321 DM322
AND P_EQ
TIM 131 #3
LD TR0
AND TIM131
OUT TR0
LD HR15.08
OR HR15.09
ANDLD
AND HR16.11
INC(38) *DM338
LD TR0
INC(38) DM252
MOV(21) #0 HR15
; rung 96
LD HR15.01
ANDNOT 35.14
OR HR15.00
OR HR15.08
ANDNOT 1.08
AND 35.15
TIM 132 #10
AND TIM132
MOV(21) #B01 DM329
; rung 97
LD HR15.03
ANDNOT 35.14
OR HR15.02
OR HR15.09
ANDNOT 1.05
AND 35.15
TIM 133 #10
AND TIM133
MOV(21) #B02 DM329
; rung 98
LD HR15.01
AND 35.14
OUT TR0
OUT 35.10
AND 1.05
TIM 134 #3
LD TR0
AND TIM134
@INC(38) DM252
MOV(21) #0 HR15

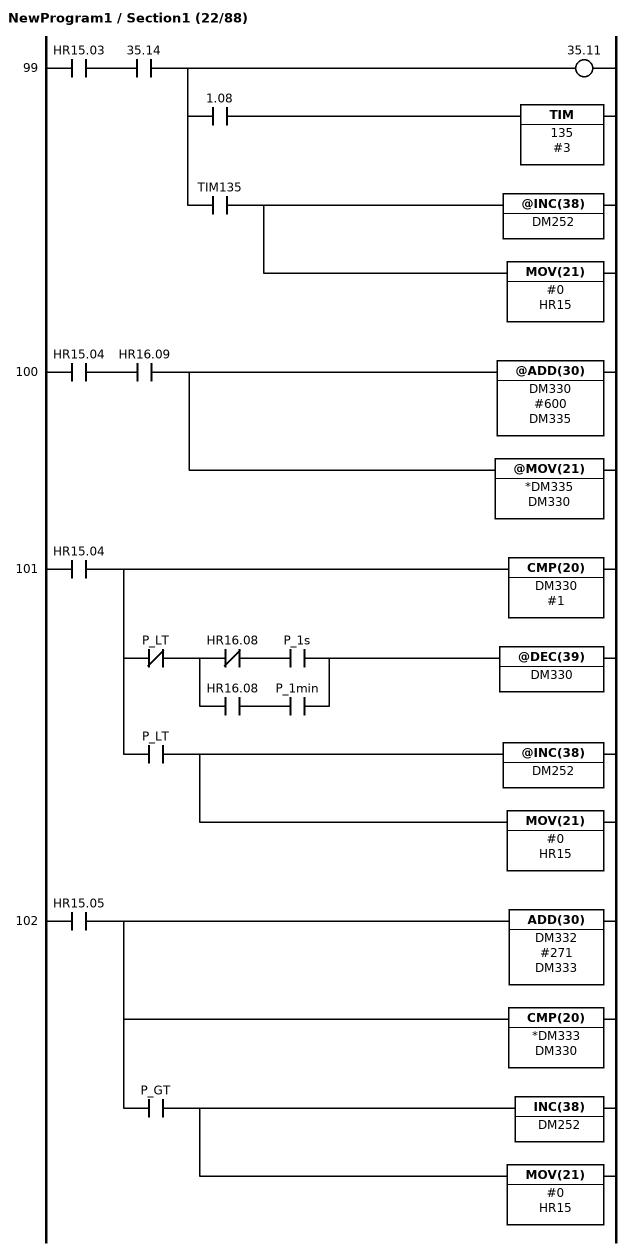
; rung 99
LD HR15.03
AND 35.14
OUT TR0
OUT 35.11
AND 1.08
TIM 135 #3
LD TR0
AND TIM135
@INC(38) DM252
MOV(21) #0 HR15
; rung 100
LD HR15.04
AND HR16.09
@ADD(30) DM330 #600 DM335
@MOV(21) *DM335 DM330
; rung 101
LD HR15.04
OUT TR0
CMP(20) DM330 #1
ANDNOT P_LT
LDNOT HR16.08
AND P_1s
LD HR16.08
AND P_1min
ORLD
ANDLD
@DEC(39) DM330
LD TR0
AND P_LT
@INC(38) DM252
MOV(21) #0 HR15
; rung 102
LD HR15.05
ADD(30) DM332 #271 DM333
CMP(20) *DM333 DM330
AND P_GT
INC(38) DM252
MOV(21) #0 HR15

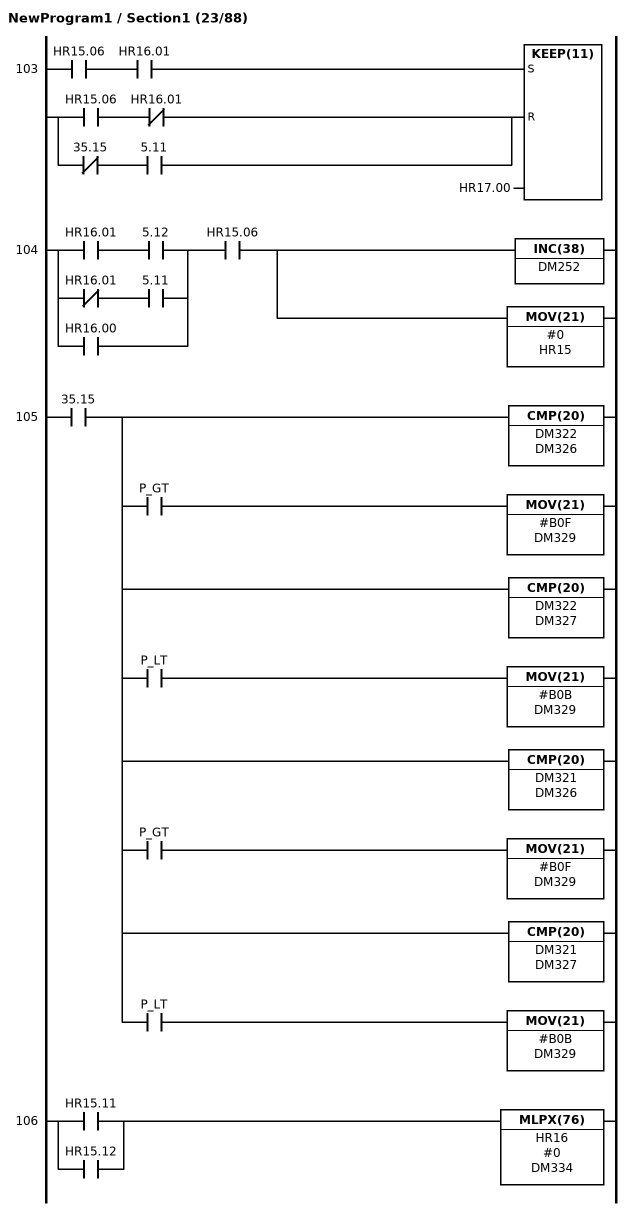
; rung 103
LD HR15.06
AND HR16.01
LD HR15.06
ANDNOT HR16.01
LDNOT 35.15
AND 5.11
ORLD
KEEP(11) HR17.00
; rung 104
LD HR16.01
AND 5.12
LDNOT HR16.01
AND 5.11
ORLD
OR HR16.00
AND HR15.06
INC(38) DM252
MOV(21) #0 HR15
; rung 105
LD 35.15
OUT TR0
CMP(20) DM322 DM326
AND P_GT
MOV(21) #B0F DM329
LD TR0
CMP(20) DM322 DM327
AND P_LT
MOV(21) #B0B DM329
LD TR0
CMP(20) DM321 DM326
AND P_GT
MOV(21) #B0F DM329
LD TR0
CMP(20) DM321 DM327
AND P_LT
MOV(21) #B0B DM329
; rung 106
LD HR15.11
OR HR15.12
MLPX(76) HR16 #0 DM334

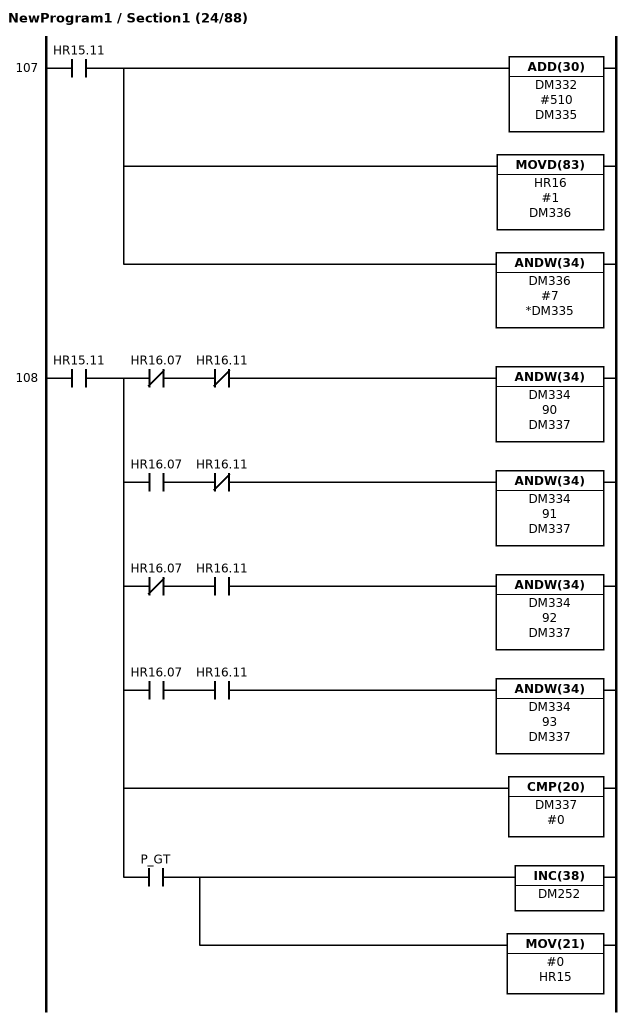
; rung 107
LD HR15.11
ADD(30) DM332 #510 DM335
MOVD(83) HR16 #1 DM336
ANDW(34) DM336 #7 *DM335
; rung 108
LD HR15.11
OUT TR0
ANDNOT HR16.07
ANDNOT HR16.11
ANDW(34) DM334 90 DM337
LD TR0
AND HR16.07
ANDNOT HR16.11
ANDW(34) DM334 91 DM337
LD TR0
ANDNOT HR16.07
AND HR16.11
ANDW(34) DM334 92 DM337
LD TR0
AND HR16.07
AND HR16.11
ANDW(34) DM334 93 DM337
LD TR0
CMP(20) DM337 #0
AND P_GT
INC(38) DM252
MOV(21) #0 HR15

